PROGRAM TestAndSet1
VAR
    nLocalBlockedCounter : DINT;
END_VAR

IF TestAndSet(GVL.bGlobalTestFlag) THEN
    (* bGlobalTestFlag was FALSE, nobody was blocking, NOW
    bGlobalTestFlag is set to TRUE and blocking others *)
    
    (* ... *)
    
    (* remove blocking by resetting the flag *) 
    GVL.bGlobalTestFlag := FALSE;
ELSE
    (* bGlobalTestFlag was TRUE, somebody is blocking *)
    nLocalBlockedCounter := nLocalBlockedCounter + 1;
    
    (* ... *)
END_IF

END_PROGRAM

(* stored: Version 1.1.0.1, ProductVersion 3.1.4024.12
   POU TestAndSet1: Id {1fbd48f8-947d-40cb-8a8d-f2473064570d}, SpecialFunc None *)
